// TIA Portal V16 export
// export: Created 2021-11-12T13:32:43.2331578Z, ExportSetting WithDefaults, DisplayName Totally Integrated Automation Portal, DisplayVersion V16 Update 3, DisplayName TIA Portal Version Control Interface, DisplayVersion V16 Update 2, DisplayName TIA Portal Openness, DisplayVersion V16 Update 3, DisplayName SINAMICS Startdrive Advanced, DisplayVersion V16 Update 5, DisplayName SINAMICS Startdrive G130, G150, S120, S150, SINAMICS MV, S210, DisplayVersion V16 Update 5, DisplayName SINAMICS Startdrive G110M, G120, G120C, G120D, G120P, G115D, DisplayVersion V16 Update 5, DisplayName STEP 7 Professional, DisplayVersion V16 Update 3, DisplayName STEP 7 Safety, DisplayVersion V16, DisplayName WinCC UA Professional, DisplayVersion V16 Update 3
DATA_BLOCK "HMI_CMD_SCH1"   // DB49
{ S7_Optimized_Access := 'TRUE' }
VERSION : 0.1
// stored: AutoNumber true, DBAccessibleFromOPCUA true, IsOnlyStoredInLoadMemory false, IsRetainMemResEnabled false, IsWriteProtectedInAS false, MemoryReserve 100
   VAR
      xxxxx___BinarySensors___xxxxx : Byte;
      xxxxx___BinaryOthers___xxxxx : Byte;
      "000UH11-SF05_22" : "UDT_CH_DI_Command";   // Blokování lisu
      "000UH10-SF12_22" : "UDT_CH_DI_Command";   // Blokování lisu
      "TT1EB01-KF02_.3" : "UDT_CH_DI_Command";   // Ohřev nástrojů 1 Kontrola chodu čerpadla
      "TT2EB01-KF02_.3" : "UDT_CH_DI_Command";   // Ohřev nástrojů 2 Kontrola chodu čerpadla
      "200CM01-BL01_14" : "UDT_CH_DI_Command";   // Jímka pod lisem Plovák nahoře Varování
      "200CM01-BL01_12" : "UDT_CH_DI_Command";   // Jímka pod lisem Plovák dole OK
      xxxxx___AnalogueSensors___xxxxx : Byte;
      "TT1EB01-KF01_29" : "UDT_CH_AI_Command";   // Tool heating 1 up actual temperature
      "TT1EB01-KF02_29" : "UDT_CH_AI_Command";   // Tool heating 1 down actual temperature
      "TT2EB01-KF01_29" : "UDT_CH_AI_Command";   // Tool heating 2 up actual temperature
      "TT2EB01-KF02_29" : "UDT_CH_AI_Command";   // Tool heating 2 down actual temperature
      xxxxx___Drives___xxxxx : Byte;
      xxxxx___Others___xxxxx : Byte;
      Commands : "UDT_SCH_Command";
      "TT1EB01-KF01_27" { S7_SetPoint := 'True'} : "UDT_CH_AO_Command";   // Setpoint tool heating 1 up
      "TT1EB01-KF02_27" : "UDT_CH_AO_Command";   // Setpoint tool heating 1 down
      "TT2EB01-KF01_27" : "UDT_CH_AO_Command";   // Setpoint tool heating 2 up
      "TT2EB01-KF02_27" : "UDT_CH_AO_Command";   // Setpoint tool heating 2 down
      xxxxx___SensorAlarms___xxxxx : Byte;
      Press : "UDT_DI_Mon_Command";   // from press
      LiveBit : "UDT_DI_Mon_Command";   // communication
      BrakeTestReqWrn : "UDT_DI_Mon_Command";   // Brake test required
      xxxxx___ProcessAlarms___xxxxx : Byte;
      "TT1EB01-KF01" : "UDT_DI_Mon_Command";   // Tool heating 1 up
      "TT1EB01-KF02" : "UDT_DI_Mon_Command";   // Tool heating 1 down
      "TT2EB01-KF01" : "UDT_DI_Mon_Command";   // Tool heating 2 up
      "TT2EB01-KF02" : "UDT_DI_Mon_Command";   // Tool heating 2 down
      "TT1EB01-KF02_3" : "UDT_DI_Mon_Command";   // Pump not running
      "TT2EB01-KF02_3" : "UDT_DI_Mon_Command";   // Pump not running
      "200CM01-BL01_15" : "UDT_DI_Mon_Command";   // Tank under press full / Jímka pod lisem Plovák nahoře Varování
      xxxxx__SafetyAlarms__xxxxx : Byte;
      ES : "UDT_DI_Mon_Command";   // E-stop
   END_VAR
BEGIN
END_DATA_BLOCK
